// SIMATIC S7-200 project (STEP 7-Micro/WIN), CPU 222 REL 01.22

ORGANIZATION_BLOCK PRINCIPAL:OB1
TITLE=COMENTARIOS DEL PROGRAMA
BEGIN
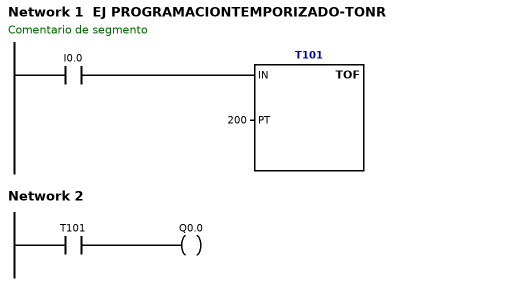
Network 1 // EJ PROGRAMACIONTEMPORIZADO-TONR

// Comentario de segmento
LD     I0.0
TOF    T101, 200
Network 2
LD     T101
=      Q0.0
END_ORGANIZATION_BLOCK
